# B&R Automation Studio project Kostka1
Automation Studio 4.1.7.61 SP

## Configuration Config1

CPU X20CP1381-RT, AutomationRuntime F4.10, Build 4.1.2, Vc V4.15.3

CPU X20CP1484, AutomationRuntime U3.09, Build 4.1.2, Vc V4.15.6

CPU X20CP1584, AutomationRuntime D4.24, Build 4.1.2, Vc V4.24.0

### Task classes (Cpu.sw)
```
Cyclic#1 (cycle 10000 us, tolerance 0 us):
  ncsdcctrl <- ncsdcctrl.prg
NcDataObjects: gAxis01a <- gAxis01obj.gAxis01a.dob, gAxis01i <- gAxis01obj.gAxis01i.dob, acp10etxen <- acp10etxen.dob, gAxis02a <- gAxis02obj.gAxis02a.dob, gAxis02i <- gAxis02obj.gAxis02i.dob
Libraries: Acp10_MC, brsystem, Acp10man, sys_lib, NcGlobal, Acp10par, Runtime, Acp10sdc, asstring
```

### Task classes (Cpu.sw)
```
Cyclic#1 (cycle 10000 us, tolerance 0 us):
  ncsdcctrl <- _MpAxis02.ncsdcctrl.prg
Cyclic#4 (cycle 100000 us, tolerance 100000 us):
  _MpAlarm <- _MpAlarm._MpAlarm.prg
  _MpAxis01 <- _MpAxis01._MpAxis01.prg
  _MpAxis02 <- _MpAxis02._MpAxis02.prg
NcDataObjects: gAxis01a <- _MpAxis01.gAxis01a.dob, gAxis01i <- _MpAxis01.gAxis01i.dob, gAxis02a <- _MpAxis02.gAxis02a.dob, acp10etxen <- acp10etxen.dob
VcDataObjects: Visu <- Visu.dob
Binaries: vccdt, vccbmp, Visu03, vccline, vcfile, arial, vccddbox, vcrt, vccstr, vcbclass, vccbtn, vcgclass, vcdsint, vcnet, vcchtml, vcmgr, vcshared, vccscale, arialbd, vccnum, vcpdvnc, vccalarm, vccurl, vccshape, vcctext, Visu01, vcpdsw, vcfntttf, vccovl, vcalarm, vcpkat, vcxml, Visu02, vcctrend, vcclbox, vccpopup, vccslider, vcdsloc, vcchspot, vcpfx20, vctcal, Config_2, Config_1, ashwd, sysconf, asfw, arconfig, Config, iomap, Acp10map, acp10cfg, Acp10sys
Libraries: Acp10_MC, brsystem, Acp10man, sys_lib, NcGlobal, Acp10par, Runtime, Acp10sdc, asstring, MpCom, MpAxis, MpAlarm, arsvcreg, astime, fileio, dataobj, powerlnk, asbrstr, asieccon, vcresman, ashw
```

### Hardware
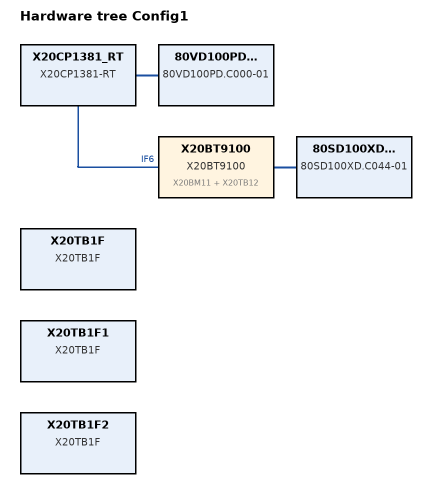
```
80SD100XD.C044-01 : 80SD100XD.C044-01 v1.8.0.0  [X2X1 -> X20BT9100.X2X1]
  BothEndSwitchesAreNormallyOpen_r1 = on
  QuickStopIsNormallyOpen_r1 = on
80VD100PD.C000-01 : 80VD100PD.C000-01 v1.1.1.1  [PLK1 -> X20CP1381_RT.IF3 (NodeNumber=1)]
  BothEndSwitchesAreNormallyOpen_r1 = on
  QuickStopIsNormallyOpen_r1 = on
X20BM11 : X20BM11 v1.0.0.0  [X2X1 -> X20CP1381_RT.IF6]
X20BT9100 : X20BT9100 v1.0.2.3  [SS1 -> X20TB12.SS; SL -> X20BM11.SL1]
X20CP1381_RT : X20CP1381-RT v1.0.2.0  [X1 -> X1.SL; X2 -> X2.SL; X3 -> X3.SL]
  Module X1 (Type=X1, Virtual=true, Version=1.0.0.0)
    Connection (Connector=SS1, TargetModule=X20TB1F, TargetConnector=SS)
    Connection (Connector=SL, TargetModule=X20CP1381_RT, TargetConnector=X1)
  Module X2 (Type=X2, Virtual=true, Version=1.0.0.0)
    Connection (Connector=SS1, TargetModule=X20TB1F1, TargetConnector=SS)
    Connection (Connector=SL, TargetModule=X20CP1381_RT, TargetConnector=X2)
  Module X3 (Type=X3, Virtual=true, Version=1.0.0.0)
    Connection (Connector=SS1, TargetModule=X20TB1F2, TargetConnector=SS)
    Connection (Connector=SL, TargetModule=X20CP1381_RT, TargetConnector=X3)
  TimerDeviceType = EPLX2X
  Cyclic1Duration = 10000
  Cyclic1Tolerance = 0
  Cyclic1Output = 1
  Cyclic2Duration = 20000
  Cyclic2Tolerance = 20000
  Cyclic3Duration = 50000
  Cyclic3Tolerance = 50000
  Cyclic4Duration = 100000
  Cyclic4Tolerance = 100000
  Cyclic5Duration = 200000
  Cyclic5Tolerance = 200000
  Cyclic6Duration = 500000
  Cyclic6Tolerance = 500000
  Cyclic7Duration = 1000000
  Cyclic7Tolerance = 1000000
  Cyclic8Duration = 10000
  Cyclic8Tolerance = 30000000
  ReActionTaskDisabled = FALSE
  TimerDevice = X20CP1381_RT.IF3
X20TB12 : X20TB12 v1.0.0.0
X20TB1F : X20TB1F v1.0.0.0
X20TB1F1 : X20TB1F v1.0.0.0
X20TB1F2 : X20TB1F v1.0.0.0
```

### Acp10map.ncm - X20CP1381_RT/Motion/Acp10map.ncm
```
NcMapping (NcSwId=Acp10)
  NcObject gAxis01 (ModuleId=80VD100PD.C000-01, Type=ncAXIS, Channel=1, AcoposSimulation=Off, InitParameter=gAxis01i, AcoposParameter=gAxis01a, Disabled=FALSE, ModuleDisabled=FALSE)
  NcObject 80VD100PD.C000-01_ncAXIS2 (ModuleId=80VD100PD.C000-01, Type=ncAXIS, Channel=2, AcoposSimulation=Off, Disabled=TRUE, ModuleDisabled=FALSE)
  NcObject 80VD100PD.C000-01_ncV_AXIS1 (ModuleId=80VD100PD.C000-01, Type=ncV_AXIS, Channel=1, Disabled=TRUE, ModuleDisabled=FALSE)
  NcObject 80VD100PD.C000-01_ncV_AXIS2 (ModuleId=80VD100PD.C000-01, Type=ncV_AXIS, Channel=2, Disabled=TRUE, ModuleDisabled=FALSE)
  NcObject gAxis02 (ModuleId=80SD100XD.C044-01, ModuleAddress=SDC_IF1.ST1, Type=ncAXIS, Channel=1, AcoposSimulation=Off, InitParameter=gAxis02i, AcoposParameter=gAxis02a, Disabled=FALSE, ModuleDisabled=FALSE)
  NcObject 80SD100XD.C044-01_ncAXIS2 (ModuleId=80SD100XD.C044-01, ModuleAddress=SDC_IF1.ST2, Type=ncAXIS, Channel=1, AcoposSimulation=Off, Disabled=TRUE, ModuleDisabled=FALSE)
```

### IoMap.iom - X20CP1584/IoMap.iom
```iecst
(********************************************************************
 * COPYRIGHT -- Bernecker + Rainer
 ********************************************************************
 * File: IoMap.iom
 * Author: vancurar
 * Created: August 06, 2015
 ********************************************************************
 * IO mapping file
 ********************************************************************)
VAR_CONFIG
	 Cyclic#1.gAxis02_DrvIf.iLifeCnt AT %IB."80SD100XD.C044-01".LifeCnt;
	 Cyclic#1.gAxis02_DrvIf.iDrvOK AT %IX."80SD100XD.C044-01".DrvOk01;
	 Cyclic#1.gAxis02_DrvIf.oBoostCurrent AT %QX."80SD100XD.C044-01".BoostCurrent01;
	 Cyclic#1.gAxis02_DrvIf.oStandStillCurrent AT %QX."80SD100XD.C044-01".StandstillCurrent01;
	 Cyclic#1.gAxis02_DrvIf.oSetTime AT %QW."80SD100XD.C044-01".SetTime01;
	 Cyclic#1.gAxis02_MotorStep0 AT %QW."80SD100XD.C044-01".Motor1Step0;
	 Cyclic#1.gAxis02_DiDoIf.iLifeCntDriveEnable AT %IB."80SD100XD.C044-01".LifeCnt;
	 Cyclic#1.gAxis02_DiDoIf.iLifeCntDriveReady AT %IB."80SD100XD.C044-01".LifeCnt;
	 Cyclic#1.gAxis02_DiDoIf.iDriveReady AT %IX."80SD100XD.C044-01".DrvOk01;
	 Cyclic#1.gAxis02_DiDoIf.oDriveEnable AT %QX."80SD100XD.C044-01".DriveEnable01;
	 Cyclic#1.gAxis02_EncIf1.iLifeCnt AT %IB."80SD100XD.C044-01".LifeCnt;
	 Cyclic#1.gAxis02_EncIf1.iEncOK AT %IX."80SD100XD.C044-01".EncOk01;
	 Cyclic#1.gAxis02_EncIf1.iActPos AT %IW."80SD100XD.C044-01".ActPos01;
	 Cyclic#1.gAxis02_EncIf1.iRefPulsePos AT %IW."80SD100XD.C044-01".RefPulsePos01;
	 Cyclic#1.gAxis02_EncIf1.iRefPulseCnt AT %IB."80SD100XD.C044-01".RefPulseCnt01;
	 Cyclic#1.gAxis02_EncIf1.iActTime AT %IW."80SD100XD.C044-01".ActTime01;
END_VAR
```

### Acp10cfg.ncc - X20CP1584/Motion/Acp10cfg.ncc
```
NcConfiguration (Version=2.49.0, NcSwId=Acp10)
  ACP10CF1_typ:
    cnt_nettrc_rec_drive = 1500
    bufsize_trace_upload = 1200
    tc_nc_man_task = Cyclic #1
    glob_pv_as_ncobject = Yes
    ncsys_dl_broadcast = Yes
    ncsys_dl_acp_reset = Yes
    safemc_log_err_to_ax = Yes
    network_init:
      ncsw_init_execute = Yes
      automatic_execute = No
      node_nr_warning = Yes
      net_err_before_ncact = Yes
    nettrc:
      enter_parsecrec = Yes
      enter_ncaction = Yes
      save_ring_startidx = Yes
    cam_prof_download:
      cam_dat_dl_parallel = No
      tc_cam_dl_parallel = Task class for NC Manager task
    plk_if[0]:
      if_name = IF3
      tc_CycDat_PLCopen = Task class for NC Manager task
      mc_broadcast_extdat = No
    sdc_if[0]:
      if_name = SDC_IF1
      mc_broadcast_size = 800
      mc_broadcast_extdat = No
```

### Acp10map.ncm - X20CP1584/Motion/Acp10map.ncm
```
NcMapping (NcSwId=Acp10, DisabledNodesAreHidden=False)
  NcObject gAxis01 (ModuleId=80VD100PD.C000-01, Type=ncAXIS, Channel=1, AcoposSimulation=Off, InitParameter=gAxis01i, AcoposParameter=gAxis01a, Disabled=FALSE, ModuleDisabled=FALSE)
  NcObject 80VD100PD.C000-01_ncAXIS2 (ModuleId=80VD100PD.C000-01, Type=ncAXIS, Channel=2, AcoposSimulation=Off, Disabled=TRUE, ModuleDisabled=FALSE)
  NcObject 80VD100PD.C000-01_ncV_AXIS1 (ModuleId=80VD100PD.C000-01, Type=ncV_AXIS, Channel=1, Disabled=TRUE, ModuleDisabled=FALSE)
  NcObject 80VD100PD.C000-01_ncV_AXIS2 (ModuleId=80VD100PD.C000-01, Type=ncV_AXIS, Channel=2, Disabled=TRUE, ModuleDisabled=FALSE)
  NcObject gAxis02 (ModuleId=80SD100XD.C044-01, ModuleAddress=SDC_IF1.ST1, Type=ncAXIS, Channel=1, AcoposSimulation=Off, AcoposParameter=gAxis02a, Disabled=FALSE, ModuleDisabled=FALSE)
  NcObject 80SD100XD.C044-01_ncAXIS2 (ModuleId=80SD100XD.C044-01, ModuleAddress=SDC_IF1.ST2, Type=ncAXIS, Channel=1, AcoposSimulation=Off, Disabled=TRUE, ModuleDisabled=FALSE)
```

### Config.mpaxisbasic - X20CP1584/mapp/Config.mpaxisbasic
```
Element gAxisBasic1 (Type=mpaxisbasic)
  AxisConfiguration = AxisWithConfiguration
    Axis:
      MovementLimits:
        PositionErrorStopLimit = 10
    Drive:
      Controller:
        LoopFilters:
          [0]
          [1]
          [2]
```

### Config_1.mpaxisbasic - X20CP1584/mapp/Config_1.mpaxisbasic
```
Element gAxisBasic2 (Type=mpaxisbasic)
  AxisConfiguration = AxisWithConfiguration
    Axis:
      BaseType = 2
      MeasurementUnit = 1
      PeriodSettings:
        Period = 1000
      MovementLimits:
        PositionErrorStopLimit = 10
    Drive:
      Gearbox:
        Input = 5
      Transformation:
        ReferenceDistance = 273
      Controller:
        LoopFilters:
          [0]
          [1]
          [2]
```

### Config_2.mpalarmbasic - X20CP1584/mapp/Config_2.mpalarmbasic
```
Element gAlarmBasic (Type=mpalarmbasic)
  mapp.Alarm.Factory:
    Reactions:
      Reaction[0]:
        Description = Example: Immediate Stop
  Alarms:
    UserAlarm:
      Alarms:
        Alarm[0]:
          Description = Example: Temperature over Tolerance
          Reaction = 1
```

## Logical view

Binary libraries used (declarations not repeated): operator, runtime, astime, AsIecCon, Acp10_MC 2.49.1, brsystem, Acp10man 2.49.1, sys_lib, NcGlobal 2.49.1, Acp10par 2.49.1, Acp10sdc 2.49.1, asstring, MpAlarm 1.20.3, MpAxis 1.20.3, MpCom 1.20.3

### Global.var - Global variables
```iecst
(********************************************************************
 * COPYRIGHT -- Bernecker + Rainer
 ********************************************************************
 * File: Global.var
 * Author: vancurar
 * Created: August 06, 2015
 ********************************************************************
 * Global variables of project Kostka1
 ********************************************************************)
VAR
	gAxis01 : ACP10AXIS_typ;
	gAxis02 : ACP10AXIS_typ;
	gAxis02_HW : SdcHwCfg_typ := (0);
	gAxis02_DrvIf : SdcDrvIf16_typ := (0);
	gAxis02_EncIf1 : SdcEncIf16_typ := (0);
	gAxis02_DiDoIf : SdcDiDoIf_typ := (0);
	gAxis02_MotorStep0 : INT := 0;
END_VAR
```


- Data object Logical/gAxis01obj/gAxis01i (Ax) (no source held here)

### Data object Logical/acp10etxen (Ett)

- acp10etxen.ett (not shown)

### Program Logical/ncsdcctrl (IEC)

#### ncsdcctrlCyclic.st
```iecst
(********************************************************************
 * COPYRIGHT -- Bernecker + Rainer
 ********************************************************************
 * Program: ncsdcctrl
 * File: ncsdcctrlCyclic.st
 * Author: vancurar
 * Created: August 06, 2015
 ********************************************************************
 * Implementation of program ncsdcctrl
 ********************************************************************)

PROGRAM _CYCLIC

(* ### BEGIN gAxis02 ### *)

(* life counter emulation of digital inputs *)
 gAxis02_DiDoIf.iLifeCntReference := gAxis02_DiDoIf.iLifeCntReference + 1;
 gAxis02_DiDoIf.iLifeCntNegHwEnd  := gAxis02_DiDoIf.iLifeCntNegHwEnd  + 1;
 gAxis02_DiDoIf.iLifeCntPosHwEnd  := gAxis02_DiDoIf.iLifeCntPosHwEnd  + 1;

(* default function model of ACOPOSmicro: convert absolute steps to delta steps - overflow save delta calculation *)
 gAxis02_MotorStep0 := gAxis02_DrvIf.oSetPos - gAxis02_oSetPosOld;
 gAxis02_oSetPosOld := gAxis02_DrvIf.oSetPos;

(* ### END gAxis02 ### *)

END_PROGRAM
```

#### ncsdcctrlInit.st
```iecst
(********************************************************************
 * COPYRIGHT -- Bernecker + Rainer
 ********************************************************************
 * Program: ncsdcctrl
 * File: ncsdcctrlInit.st
 * Author: vancurar
 * Created: August 06, 2015
 ********************************************************************
 * Implementation of program ncsdcctrl
 ********************************************************************)

PROGRAM _INIT

(* ### BEGIN gAxis02 ### *)

(* initialize general interfaces *)
 gAxis02.size := gAxis02.size;
 gAxis02_HW.DrvIf_Typ := ncSDC_DRVSM16;
 strcpy( ADR(gAxis02_HW.DrvIf_Name[0]), ADR('gAxis02_DrvIf') );
 gAxis02_HW.DiDoIf_Typ := ncSDC_DIDO;
 strcpy( ADR(gAxis02_HW.DiDoIf_Name[0]), ADR('gAxis02_DiDoIf') );
 gAxis02_HW.EncIf1_Typ := ncSDC_ENC16;
 strcpy( ADR(gAxis02_HW.EncIf1_Name[0]), ADR('gAxis02_EncIf1') );
 gAxis02_EncIf1.iLifeCnt := gAxis02_EncIf1.iLifeCnt;

(* initialize old-value for delta step calculation *)
 gAxis02_oSetPosOld := gAxis02_DrvIf.oSetPos;

(* ### END gAxis02 ### *)

END_PROGRAM
```

#### ncsdcctrl.var
```iecst
(********************************************************************
 * COPYRIGHT -- Bernecker + Rainer
 ********************************************************************
 * Program: ncsdcctrl
 * File: ncsdcctrl.var
 * Author: vancurar
 * Created: August 06, 2015
 ********************************************************************
 * Local variables of program ncsdcctrl
 ********************************************************************)
VAR
	gAxis02_oSetPosOld : INT := 0;
END_VAR
```

### Package Logical/gAxis02obj - gAxis02obj

- Data object Logical/gAxis02obj/gAxis02a (Apt) (no source held here)

### Data object Logical/gAxis02obj/gAxis02i (Ax)

#### gAxis02i.ax
```
InitParameter (Version=2.49.1, NcSwId=ACP10)
  ACP10AXIS_typ:
    dig_in:
      level:
        reference = ncACTIV_HI
        pos_hw_end = ncACTIV_HI
        neg_hw_end = ncACTIV_HI
        trigger1 = ncACTIV_HI
        trigger2 = ncACTIV_HI
    encoder_if:
      parameter:
        count_dir = ncSTANDARD
        scaling:
          load:
            units = 1000
            rev_motor = 1
    limit:
      parameter:
        v_pos = 10000.0
        v_neg = 10000.0
        a1_pos = 50000.0
        a2_pos = 50000.0
        a1_neg = 50000.0
        a2_neg = 50000.0
        t_jolt = 0.0
        t_in_pos = 0.0
        pos_sw_end = 8388607
        neg_sw_end = -8388608
        ds_warning = 500.0
        ds_stop = 1000.0
        a_stop = 1.0e+30
        dv_stop = 0.0
        dv_stop_mode = ncOFF
    controller:
      mode = ncPOSITION
      position:
        kv = 50.0
        tn = 0.0
        t_predict = 0.05
        t_total = 0.05
        p_max = 1.0e+30
        i_max = 0.0
      speed:
        kv = 2.0
        tn = 0.0
        t_filter = 0.0
        isq_filter1:
          type = ncOFF
          a0 = 0.0
          a1 = 0.0
          b0 = 0.0
          b1 = 0.0
          b2 = 0.0
          c0_par_id = 0
          c1_par_id = 0
        isq_filter2:
          type = ncOFF
          a0 = 0.0
          a1 = 0.0
          b0 = 0.0
          b1 = 0.0
          b2 = 0.0
          c0_par_id = 0
          c1_par_id = 0
        isq_filter3:
          type = ncOFF
          a0 = 0.0
          a1 = 0.0
          b0 = 0.0
          b1 = 0.0
          b2 = 0.0
          c0_par_id = 0
          c1_par_id = 0
      uf:
        type = ncLINEAR
        auto_config = ncMOTOR_PAR
        u0 = 0.0
        un = 0.0
        fn = 50.0
        k_f_slip = 0.0
      ff:
        torque_load = 0.0
        torque_pos = 0.0
        torque_neg = 0.0
        kv_torque = 0.0
        inertia = 0.0
        t_filter_a = 0.0
    move:
      stop:
        parameter[0]:
          decel_ramp = ncA_LIMIT
          controller = ncON
        parameter[1]:
          decel_ramp = ncA_LIMIT
          controller = ncON
        parameter[2]:
          decel_ramp = ncA_LIMIT
          controller = ncON
        parameter[3]:
          decel_ramp = ncA_LIMIT
          controller = ncON
        quickstop:
          decel_ramp = ncA_LIMIT
        drive_error:
          decel_ramp = ncA_LIMIT
      homing:
        parameter:
          s = 0
          v_switch = 5000.0
          v_trigger = 500.0
          a = 50000.0
          mode = ncDIRECT
          edge_sw = ncPOSITIVE
          start_dir = ncPOSITIVE
          trigg_dir = ncPOSITIVE
          ref_pulse = ncOFF
          fix_dir = ncOFF
          tr_s_block = 0.0
          torque_lim = 0.0
          ds_block = 0.0
          ds_stop = 0.0
      basis:
        parameter:
          v_pos = 5000.0
          v_neg = 5000.0
          a1_pos = 50000.0
          a2_pos = 50000.0
          a1_neg = 50000.0
          a2_neg = 50000.0
    message:
      text:
        parameter:
          format = ncBREAK
          columns = 80
          data_modul = acp10etxen
```

### _MpAlarmGlobal.var
```iecst
VAR
	MainAlarmUIConnect : MpAlarmBasicUIConnect100Type; (*Structure contains Alarm, Acknowledge and AddInfo arrays for VC4*)
END_VAR
```

### Program Logical/_MpAlarm/_MpAlarm (IEC)

#### Variables.var
```iecst
VAR
	MpAlarmBasic_0 : MpAlarmBasic;
	MpAlarmBasicUI_Main : MpAlarmBasicUI;
	MpAlarmBasicUISetupMain : MpAlarmBasicUISetupType;
	MpAlarmBasicUI_Axis1 : MpAlarmBasicUI;
	MpAlarmBasicUISetupAxis1 : MpAlarmBasicUISetupType;
	MpAlarmBasicUI_Axis2 : MpAlarmBasicUI;
	MpAlarmBasicUISetupAxis2 : MpAlarmBasicUISetupType;
	simMainAlarmIndex : INT;
END_VAR
```

#### Cyclic.st
```iecst
PROGRAM _CYCLIC

	// MpAlarm FB call
	MpAlarmBasic_0(MpLink := ADR(gAlarmBasic), Enable := 1);

	(*	TESTING OF ALARM SET/RESET
		Setting 'i' or ('j') var to nonzero value leads to set alarm on index 'i - 1' ('j - 1') in case that 'i' ('j') is greater than 0 and to reset in similar way in case that 'i'('j') is lower than 0
		Setting 'k'('l') to nonzero value leads to set user alarm on index 15 in case that 'k'('l') is greater than 0 and to reset this alarm in case that 'k'('l') is lower than 0
	*)

	// Set/Reset alarm on i-1 th index in gMain (if i > 100, there is no influence to MpAlarmBasic)
	IF simMainAlarmIndex > 0 THEN
		MpAlarmSet(gAlarmBasic, simMainAlarmIndex - 1,'addInfo');
	ELSIF simMainAlarmIndex < 0 THEN
		MpAlarmReset(gAlarmBasic, -(simMainAlarmIndex + 1));
	END_IF

END_PROGRAM
```

#### Init.st
```iecst
PROGRAM _INIT

	//MpAxis2AlarmUIConnect is MpAlarmBasicUIConnect200Type (user defined) because there is 200 user alarms
	MpAlarmBasicUISetupMain.AcknowledgeImage := ADR(MainAlarmUIConnect.AcknowledgeImage);
	MpAlarmBasicUISetupMain.AddInfo := ADR(MainAlarmUIConnect.AddInfo);
	MpAlarmBasicUISetupMain.AddInfoStringSize := SIZEOF(MainAlarmUIConnect.AddInfo[0]);
	MpAlarmBasicUISetupMain.AlarmImage := ADR(MainAlarmUIConnect.AlarmImage);
	MpAlarmBasicUISetupMain.ImageSize := SIZEOF(MainAlarmUIConnect.AlarmImage);

	//MpAlarmBasicUI FB init settings
	MpAlarmBasicUI_Main.MpLink := ADR(gAlarmBasic);
	MpAlarmBasicUI_Main.Mode := mpALARM_BASIC_UI_MODE_USER;
	MpAlarmBasicUI_Main.UISetup := MpAlarmBasicUISetupMain;

END_PROGRAM
```

### _MpAxis01Global.var
```iecst
VAR
	Axis01Par : MpAxisBasicParType; (*mapp Axis 1 parameters*)
	gAxis01 : ACP10AXIS_typ; (*ACP10 axis*)
	MpAxis1AlarmUIConnect : MpAlarmBasicUIConnect20Type; (*Structure contains Alarm, Acknowledge and AddInfo arrays for VC4*)
	MpAxisBasic_Axis1 : MpAxisBasic; (*mapp Axis component for Axis1*)
END_VAR
```

- Data object Logical/_MpAxis01/gAxis01a (Apt) (no source held here)

### Data object Logical/_MpAxis01/gAxis01i (Ax)

#### gAxis01i.ax
```
InitParameter (Version=2.49.1, NcSwId=ACP10)
  ACP10AXIS_typ:
    dig_in:
      level:
        reference = ncACTIV_HI
        pos_hw_end = ncACTIV_HI
        neg_hw_end = ncACTIV_HI
        trigger1 = ncACTIV_HI
        trigger2 = ncACTIV_HI
    encoder_if:
      parameter:
        count_dir = ncSTANDARD
        scaling:
          load:
            units = 1000
            rev_motor = 1
    limit:
      parameter:
        v_pos = 10000.0
        v_neg = 10000.0
        a1_pos = 50000.0
        a2_pos = 50000.0
        a1_neg = 50000.0
        a2_neg = 50000.0
        t_jolt = 0.0
        t_in_pos = 0.0
        pos_sw_end = 8388607
        neg_sw_end = -8388608
        ds_warning = 500.0
        ds_stop = 1000.0
        a_stop = 1.0e+30
        dv_stop = 0.0
        dv_stop_mode = ncOFF
    controller:
      mode = ncPOSITION
      position:
        kv = 400.0
        tn = 0.0
        t_predict = 0.0004
        t_total = 0.0004
        p_max = 1.0e+30
        i_max = 0.0
      speed:
        kv = 0.05
        tn = 0.0
        t_filter = 0.0
        isq_filter1:
          type = ncNOTCH
          a0 = 430.528
          a1 = 400.0
          b0 = 0.0
          b1 = 0.0
          b2 = 0.0
          c0_par_id = 0
          c1_par_id = 0
        isq_filter2:
          type = ncOFF
          a0 = 0.0
          a1 = 0.0
          b0 = 0.0
          b1 = 0.0
          b2 = 0.0
          c0_par_id = 0
          c1_par_id = 0
        isq_filter3:
          type = ncOFF
          a0 = 0.0
          a1 = 0.0
          b0 = 0.0
          b1 = 0.0
          b2 = 0.0
          c0_par_id = 0
          c1_par_id = 0
      uf:
        type = ncLINEAR
        auto_config = ncMOTOR_PAR
        u0 = 0.0
        un = 0.0
        fn = 50.0
        k_f_slip = 0.0
      ff:
        torque_load = 0.0
        torque_pos = 0.0
        torque_neg = 0.0
        kv_torque = 0.0
        inertia = 0.0
        t_filter_a = 0.0
    move:
      stop:
        parameter[0]:
          decel_ramp = ncA_LIMIT
          controller = ncON
        parameter[1]:
          decel_ramp = ncA_LIMIT
          controller = ncON
        parameter[2]:
          decel_ramp = ncA_LIMIT
          controller = ncON
        parameter[3]:
          decel_ramp = ncA_LIMIT
          controller = ncON
        quickstop:
          decel_ramp = ncA_LIMIT
        drive_error:
          decel_ramp = ncA_LIMIT
      homing:
        parameter:
          s = 0
          v_switch = 5000.0
          v_trigger = 500.0
          a = 50000.0
          mode = ncDIRECT
          edge_sw = ncPOSITIVE
          start_dir = ncPOSITIVE
          trigg_dir = ncPOSITIVE
          ref_pulse = ncOFF
          fix_dir = ncOFF
          tr_s_block = 0.0
          torque_lim = 0.0
          ds_block = 0.0
          ds_stop = 0.0
      basis:
        parameter:
          v_pos = 5000.0
          v_neg = 5000.0
          a1_pos = 50000.0
          a2_pos = 50000.0
          a1_neg = 50000.0
          a2_neg = 50000.0
    message:
      text:
        parameter:
          format = ncBREAK
          columns = 80
          data_modul = acp10etxen
```

### Program Logical/_MpAxis01/_MpAxis01 (IEC)

#### Variables.var
```iecst
VAR
	MpAlarmBasicUI_Axis1 : MpAlarmBasicUI;
	MpAlarmBasicUISetupAxis1 : MpAlarmBasicUISetupType;
END_VAR
```

#### Cyclic.st
```iecst
PROGRAM _CYCLIC

	//Technological mapp FB call
	MpAxisBasic_Axis1();

	//FBs MpAlarmUI for VC4 visualization
	MpAlarmBasicUI_Axis1.Enable := MpAxisBasic_Axis1.Active;
	MpAlarmBasicUI_Axis1();

END_PROGRAM
```

#### Init.st
```iecst
PROGRAM _INIT

	//mapp FBs basic init settings
	MpAxisBasic_Axis1.MpLink := ADR(gAxisBasic1);
	MpAxisBasic_Axis1.Axis := ADR(gAxis01);
	MpAxisBasic_Axis1.Parameters := ADR(Axis01Par);
	MpAxisBasic_Axis1.Enable := 1;

	//MpAxis1AlarmUIConnect is MpAlarmBasicUIConnect20Type because there is only 14 MpAxis alarms and one user alarm
	MpAlarmBasicUISetupAxis1.AcknowledgeImage := ADR(MpAxis1AlarmUIConnect.AcknowledgeImage);
	MpAlarmBasicUISetupAxis1.AddInfo := ADR(MpAxis1AlarmUIConnect.AddInfo);
	MpAlarmBasicUISetupAxis1.AddInfoStringSize := SIZEOF(MpAxis1AlarmUIConnect.AddInfo[0]);
	MpAlarmBasicUISetupAxis1.AlarmImage := ADR(MpAxis1AlarmUIConnect.AlarmImage);
	MpAlarmBasicUISetupAxis1.ImageSize := SIZEOF(MpAxis1AlarmUIConnect.AlarmImage);

	//MpAlarmBasicUI FB init settings
	MpAlarmBasicUI_Axis1.MpLink := ADR(gAxisBasic1);
	MpAlarmBasicUI_Axis1.Mode := mpALARM_BASIC_UI_MODE_ALL;
	MpAlarmBasicUI_Axis1.UISetup := MpAlarmBasicUISetupAxis1;

END_PROGRAM
```

### _MpAxis02Global.var
```iecst
VAR
	Axis02Par : MpAxisBasicParType; (*mapp Axis 2 parameters*)
	gAxis02 : ACP10AXIS_typ;
	gAxis02_DiDoIf : SdcDiDoIf_typ := (0);
	gAxis02_DrvIf : SdcDrvIf16_typ := (0);
	gAxis02_EncIf1 : SdcEncIf16_typ := (0);
	gAxis02_HW : SdcHwCfg_typ := (0);
	gAxis02_MotorStep0 : INT := 0;
	MpAxis2AlarmUIConnect : MpAlarmBasicUIConnect20Type; (*Structure contains Alarm, Acknowledge and AddInfo arrays for VC4*)
	MpAxisBasic_Axis2 : MpAxisBasic; (*mapp Axis component for Axis2*)
END_VAR
```

### Data object Logical/_MpAxis02/gAxis02a (Apt)

#### gAxis02a.apt
```
AcoposParameterTable:
  Root Parameters:
    64232 = 51200 (Name=SM_SCALE_STEP)
    64233 = 27300 (Name=SM_SCALE_LOAD_UNITS)
    64234 = 5 (Name=SM_SCALE_LOAD_MOTREV)
    109 = 1024 (Name=SCALE_ENCOD_INCR)
    230 = PCTRL_S_SET (Name=PCTRL_S_ACT_PARID, Disabled=TRUE)  // CTRL Position controller: Actual encoder position parameter ID
```

### Program Logical/_MpAxis02/_MpAxis02 (IEC)

#### Init.st - Init code
```iecst
PROGRAM _INIT

	MpAxisBasic_Axis2.MpLink := ADR(gAxisBasic2);
	MpAxisBasic_Axis2.Axis := ADR(gAxis02);
	MpAxisBasic_Axis2.Parameters := ADR(Axis02Par);
	MpAxisBasic_Axis2.Enable := 1;

	//MpAxis2AlarmUIConnect is MpAlarmBasicUIConnect20Type because there is only 14 MpAxis alarms and one user alarm
	MpAlarmBasicUISetupAxis2.AcknowledgeImage := ADR(MpAxis2AlarmUIConnect.AcknowledgeImage);
	MpAlarmBasicUISetupAxis2.AddInfo := ADR(MpAxis2AlarmUIConnect.AddInfo);
	MpAlarmBasicUISetupAxis2.AddInfoStringSize := SIZEOF(MpAxis2AlarmUIConnect.AddInfo[0]);
	MpAlarmBasicUISetupAxis2.AlarmImage := ADR(MpAxis2AlarmUIConnect.AlarmImage);
	MpAlarmBasicUISetupAxis2.ImageSize := SIZEOF(MpAxis2AlarmUIConnect.AlarmImage);

	//MpAlarmBasicUI FB init settings
	MpAlarmBasicUI_Axis2.MpLink := ADR(gAxisBasic2);
	MpAlarmBasicUI_Axis2.Mode := mpALARM_BASIC_UI_MODE_ALL;
	MpAlarmBasicUI_Axis2.UISetup := MpAlarmBasicUISetupAxis2;

END_PROGRAM
```

#### Cyclic.st - Cyclic code
```iecst
PROGRAM _CYCLIC

	//Technological mapp FB call
	MpAxisBasic_Axis2();

	//FBs MpAlarmUI for VC4 visualization
	MpAlarmBasicUI_Axis2.Enable := MpAxisBasic_Axis2.Active;
	MpAlarmBasicUI_Axis2();

END_PROGRAM
```

#### Variables.var - Local variables
```iecst
VAR
	MpAlarmBasicUI_Axis2 : MpAlarmBasicUI;
	MpAlarmBasicUISetupAxis2 : MpAlarmBasicUISetupType;
END_VAR
```

- Program Logical/_MpAxis02/ncsdcctrl (IEC) (no source held here)

Listed in the project but not available here: Logical/gAxis01obj/gAxis01a, Logical/ncsdcctrl/ncsdcctrl.typ, Logical/_MpAxis02/ncsdcctrl/ncsdcctrlCyclic.st, Logical/_MpAxis02/ncsdcctrl/ncsdcctrlInit.st, Logical/_MpAxis02/ncsdcctrl/ncsdcctrl.var
